FUNCTION_BLOCK F_Calc
VAR_INPUT
	nGetal : INT := 0;
END_VAR
VAR_OUTPUT
	
END_VAR
VAR
	_fAns : REAL;
	_fSavedValue : REAL;
END_VAR

PROPERTY PUBLIC fAns : REAL
GET
fAns := _fAns;
END_GET
END_PROPERTY

PROPERTY PUBLIC fSavedValue : REAL
GET
fSavedValue := _fSavedValue;
END_GET
SET
VAR
	//fGetal : REAL;
END_VAR
_fSavedValue := fSavedValue;
END_SET
END_PROPERTY

METHOD PUBLIC M_Add : REAL
VAR_INPUT
		getalOmOpTeTellen : REAL ;
END_VAR
_fAns := _fAns + getalOmOpTeTellen;
END_METHOD

METHOD PUBLIC M_Divide : REAL
VAR_INPUT
		GetalOmTeDelen : REAL;
END_VAR
_fAns := _fAns / GetalOmTeDelen;
END_METHOD

METHOD PUBLIC M_Multiply : REAL
VAR_INPUT
	GetalOmTeVermenigvuldigen : REAL;
END_VAR
_fAns := _fAns * GetalOmTeVermenigvuldigen;
END_METHOD

METHOD PUBLIC M_Save
VAR_INPUT
END_VAR
_fSavedValue := _fAns;
END_METHOD

METHOD PUBLIC M_Subtract : REAL
VAR_INPUT
	getalOmAfTeTrekken : REAL;
END_VAR
_fAns := _fAns - getalOmAfTeTrekken;
END_METHOD

END_FUNCTION_BLOCK

(* stored: Version 1.1.0.1, ProductVersion 3.1.4024.13
   POU F_Calc: Id {f8a72b7c-41b2-461a-bd0c-4813f483d062}, SpecialFunc None
   Property fAns: Id {29aa46e8-2a56-4b92-84e2-63b01c8e76f2}
   Get Get: Id {cedb09b0-411e-4f47-beab-5e1ea1270014}
   Property fSavedValue: Id {a7fd3f70-aa0b-4693-8c99-5a1e754fa38d}
   Get Get: Id {992703e8-8292-436e-a4aa-d77b7a671e64}
   Set Set: Id {abe5e5ae-17ee-45c8-ba18-b725a6e28db0}
   Method M_Add: Id {ccb8c972-52af-4245-a034-9ba4cd3b4fc1}
   Method M_Divide: Id {ceaec26a-7484-45c7-ae16-e33819cbdc3c}
   Method M_Multiply: Id {f6932f9c-a959-40f5-957f-8548bc23edfc}
   Method M_Save: Id {1f363065-0c6e-44f5-9b38-78905070f6f4}
   Method M_Subtract: Id {141b6fa8-96b4-4383-85c6-529bc8ebf37f} *)
